// TwinCAT 3 PLC project PLC
// ProgramVersion: 3.1.4024.0
// libraries:
//   Tc2_Standard, * (Beckhoff Automation GmbH)
//   Tc2_System, * (Beckhoff Automation GmbH)
//   Tc2_Utilities, * (Beckhoff Automation GmbH)
//   Tc3_JsonXml, * (Beckhoff Automation GmbH)
//   Tc3_Module, * (Beckhoff Automation GmbH)
// project tree:
//   / FB_DynamicArrayBase64.TcPOU, FB_DynamicArrayBinary.TcPOU, FB_DynamicArrayOfLREAL.TcPOU, FB_DynamicArrayOfInt.TcPOU, MAIN.TcPOU, PlcTask.TcTTO
//   Test/ FB_Test.TcPOU, I_Test.TcIO
//   Utilities/ FB_TimeLimitedIterator.TcPOU
// real-time tasks:
//   TASK PlcTask: cycle T#10ms, priority 20, ADS port 350

CONFIGURATION PLC
    RESOURCE PLC ON TwinCAT3
        TASK PlcTask(INTERVAL := T#10ms, PRIORITY := 20);
        PROGRAM MAIN WITH PlcTask : MAIN;
    END_RESOURCE
END_CONFIGURATION

// ---- Test/I_Test.TcIO
INTERFACE I_Test

METHOD METH : BOOL
VAR_INPUT
END_VAR
END_METHOD

PROPERTY Name : String
GET
END_GET
END_PROPERTY

END_INTERFACE

// ---- MAIN.TcPOU
PROGRAM MAIN
VAR
	aArray : FB_DynamicArrayBase64;
	bRemoveLast: BOOL;
	bRemoveFirst : BOOL;
	bRemoveIndex : BOOL;
	
	bAddTest : BOOL;
	bAddTestLoop : BOOL;
	bClear : BOOL;
	
	bSetIndex : BOOL;
END_VAR
VAR
	//=============================
	// Remove Index Test
	RemoveIndex : UDINT;
	
	//=============================
	// Set Inex Test
	nSetIndex : UDINT;
	//=============================
	// Add Test
	WriteBool : BOOL;
	WriteReal : LREAL;
	WriteString : STRING;
	
	iTest : I_Test;
	fbTest : FB_Test;
	
	//=============================
	// Add Test Loop
	nAddTest : INT := 1000;
	i : INT;
	sTest : STRING(32766);
	
	ArrayElements : UDINT;
	
	
	//==================================================
	//Get
	ReadBOOL : BOOL;
	ReadReal : LREAL;
	ReadString : STRING;
	ReadInterface : I_Test;
	
	bReadBOOL : BOOL;
	bReadREAL : BOOL;
	bReadString : BOOL;
	bReadInterface : BOOL;
	ReadIndex : UDINT;
	//==================================================
	//Time
	fbTimeLimitedIterator : FB_TimeLimitedIterator := (TaskUsagePercent := 100);
	ReadTime : LTIME;
	
	aTime : ARRAY[0..100000] OF LINT;
	aLREAL : FB_DynamicArrayOfINT;
	nTestLoop : UDINT := 10000;
	f : UDINT;
	fReadWrite : LINT;
	
	tTimeWriteArray : LTIME;
	tTimeReadArray : LTIME;
	
	tTimeAddDynamicArray : LTIME;
	tTimeWriteDynamicArray : LTIME;
	tTimeReadDynamicArray : LTIME;
	
	WriteFaktor : LREAL;
	ReadFaktor : LREAL;
END_VAR

ArrayElements := aArray.Count;
iTest := fbTest;

//=============================
// Add Test
IF bAddTest THEN
	bAddTest := FALSE;	
	aArray.AddLast(WriteBool);
	aArray.AddLast(WriteReal);
	aArray.AddStringLast(WriteString);
	aArray.AddLast(iTest);
END_IF

//=============================
// Add Test
IF bSetIndex THEN
	bSetIndex := FALSE;	
	aArray.TrySetIndex(nSetIndex, WriteBool);

END_IF
//=============================
// Add Test Loop
	IF bAddTestLoop THEN
		bAddTestLoop := FALSE;
		IF nAddTest > 0 THEN
			FOR i := 0 TO nAddTest - 1 DO
				aArray.AddLast(WriteBool);
				aArray.AddLast(WriteReal);
				aArray.AddStringLast(WriteString);
				aArray.AddLast(iTest);
			END_FOR
		END_IF
	END_IF

//=============================
// Clear
	IF bClear THEN
		bClear := FALSE;
		aArray.Clear();
	END_IF

//=============================
// Remove
	IF bRemoveLast THEN
		bRemoveLast := FALSE;
		aArray.RemoveLast();
	END_IF
	IF bRemoveFirst THEN
		bRemoveFirst := FALSE;
		aArray.RemoveFirst();
	END_IF
	IF bRemoveIndex THEN
		bRemoveIndex := FALSE;
		aArray.TryDeleteIndex(RemoveIndex);
	END_IF
	
//==================================================
//Get

	fbTimeLimitedIterator.SetIterationStartTime();
	
	bReadBOOL := aArray.TryGetIndex(ReadIndex,ReadBool);
	bReadREAL := aArray.TryGetIndex(ReadIndex,ReadReal);
	bReadString := aArray.TryGetIndex(ReadIndex,ReadString);
	bReadInterface := aArray.TryGetIndex(ReadIndex, ReadInterface);
	
	ReadTime := fbTimeLimitedIterator.CurrentIterationTime();

//==========================================================
// Debug String
	aArray.CopyArrayString(pDoc:= sTest, nDoc := SIZEOF(sTest));
	
//==========================================================
// Timing Test
	nTestLoop := LIMIT(0,nTestLoop ,100000);
	
	fbTimeLimitedIterator.SetIterationStartTime();
		FOR f := 0 TO nTestLoop DO
			aTime[f] := fReadWrite;
		END_FOR
	tTimeWriteArray := fbTimeLimitedIterator.CurrentIterationTime();
	
	
	fbTimeLimitedIterator.SetIterationStartTime();
		FOR f := 0 TO nTestLoop DO
			fReadWrite := aTime[f];
		END_FOR
	tTimeReadArray := fbTimeLimitedIterator.CurrentIterationTime();
	

	
	aLREAL.Clear();
	
	fbTimeLimitedIterator.SetIterationStartTime();
		FOR f := 0 TO nTestLoop DO
			aLREAL.AddLast(fReadWrite);
		END_FOR
	tTimeAddDynamicArray := fbTimeLimitedIterator.CurrentIterationTime();
	
	fbTimeLimitedIterator.SetIterationStartTime();
		FOR f := 0 TO nTestLoop DO
			aLREAL.TrySetIndex(f,fReadWrite);
		END_FOR
	tTimeWriteDynamicArray := fbTimeLimitedIterator.CurrentIterationTime();
	
	fbTimeLimitedIterator.SetIterationStartTime();
		FOR f := 0 TO nTestLoop DO
			aLREAL.TryGetIndex(f,fReadWrite);
		END_FOR
	tTimeReadDynamicArray := fbTimeLimitedIterator.CurrentIterationTime();

	
	
	IF tTimeReadArray <> LTIME#0S THEN
		ReadFaktor := TO_LREAL(TO_LREAL(tTimeReadDynamicArray*10000)/TO_LREAL(tTimeReadArray*10000));
	END_IF
	IF tTimeWriteArray <> LTIME#0S THEN
		WriteFaktor := TO_LREAL(TO_LREAL(tTimeWriteDynamicArray*10000)/TO_LREAL( tTimeWriteArray*10000));
	END_IF

END_PROGRAM

// ---- FB_DynamicArrayBase64.TcPOU
{attribute 'no_explicit_call' := 'This FB is a CLASS and must be accessed using methods or properties'}
{attribute 'enable_dynamic_creation'}
{attribute 'hide_all_locals'}
FUNCTION_BLOCK FB_DynamicArrayBase64
VAR
	buffer : FB_JsonDynDomParser;
	root : sJsonValue;
END_VAR

PROPERTY PRIVATE _Array : sJsonValue
GET
IF root <> 0 THEN
	_Array := root;
ELSE
	root := buffer.NewDocument();
	_Array := buffer.SetArray(root,0);
END_IF
END_GET
END_PROPERTY

METHOD PUBLIC AddLast : BOOL
VAR_INPUT
	Value : ANY;
END_VAR
AddLast := buffer.PushbackBase64Value(v:= _Array, p := Value.pValue,n := Value.diSize) <> 0;
END_METHOD

METHOD PUBLIC AddStringLast : BOOL
VAR_INPUT
	Value : ANY_STRING;
END_VAR
AddStringLast := buffer.PushbackBase64Value(v:= _Array, p := Value.pValue,n := TO_DINT(LEN2(Value.pValue)+ 1)) <> 0;
END_METHOD

METHOD PUBLIC Clear : BOOL
VAR
	_arrayElement : SJsonAIterator;
END_VAR
_arrayElement := buffer.ArrayBegin(_array);
IF _arrayElement <> 0 THEN
	Clear := buffer.ClearArray(v := _array,i := _arrayElement);
END_IF
END_METHOD

METHOD PUBLIC CopyArrayString : BOOL
VAR_IN_OUT CONSTANT
  	pDoc : STRING; 
END_VAR
VAR_INPUT
	nDoc : UDINT;
END_VAR
CopyArrayString := buffer.copyjson(v:= _Array, pDoc:= pDoc,nDoc := nDoc) <> 0;
END_METHOD

PROPERTY PUBLIC Count : UDINT
GET
Count := buffer.GetArraySize(_array);
END_GET
END_PROPERTY

PROPERTY PUBLIC FirstIndex : UDINT
GET
FirstIndex := 0;
END_GET
END_PROPERTY

PROPERTY PUBLIC LastIndex : UDINT
GET
IF Count = 0 THEN
	LastIndex := 0;
ELSE 
	LastIndex := Count - 1;
END_IF
END_GET
END_PROPERTY

METHOD PUBLIC RemoveFirst : BOOL
VAR
	_arrayElement : SJsonAIterator;
END_VAR
RemoveFirst := TryDeleteIndex(0);
END_METHOD

METHOD PUBLIC RemoveLast: BOOL
VAR
	_arrayElement : SJsonAIterator;
END_VAR
RemoveLast := TryDeleteIndex(LastIndex);
END_METHOD

METHOD PUBLIC TryDeleteIndex : BOOL
VAR_INPUT
	Index : UDINT;
END_VAR
VAR
	_arrayElement : SJsonAIterator;
END_VAR
_arrayElement := buffer.GetArrayValueByIdx(_Array, Index);
IF _arrayElement <> 0 THEN
	TryDeleteIndex := buffer.RemoveArray(v := _array,i := _arrayElement);
END_IF
END_METHOD

METHOD PUBLIC TryGetIndex : BOOL;
VAR_INPUT
	Index : UDINT;
	Destination : ANY;
END_VAR
TryGetIndex := buffer.GetBase64(v:=  buffer.GetArrayValueByIdx(_Array, Index),p := Destination.pValue, n:= Destination.diSize) <> 0;
END_METHOD

METHOD PUBLIC TryGetIndexTo : BOOL;
VAR_INPUT
	Index : UDINT;
	Destination : PVOID;
	DestinationSize : UDINT;
END_VAR
VAR
	_arrayElement : SJsonAIterator;
END_VAR
_arrayElement := buffer.GetArrayValueByIdx(_Array, Index);
IF _arrayElement <> 0 THEN
	TryGetIndexTo := buffer.GetBase64(v:= _arrayElement,p := Destination, n:= TO_DINT(DestinationSize)) <> 0;
END_IF
END_METHOD

METHOD PUBLIC TrySetIndex : BOOL
VAR_INPUT
	Index : UDINT;
	Value : ANY;
END_VAR
TrySetIndex := buffer.SetBase64(v:= buffer.GetArrayValueByIdx(_Array, Index),p := Value.pValue, n:= Value.diSize) <> 0;
END_METHOD

METHOD PUBLIC TrySetIndexTo : BOOL
VAR_INPUT
	Index : UDINT;
	Value : PVOID;
	ValueSize : UDINT;
END_VAR
VAR
	_arrayElement : SJsonAIterator;
END_VAR
_arrayElement := buffer.GetArrayValueByIdx(_Array, Index);
IF _arrayElement <> 0 THEN
	TrySetIndexTo := buffer.SetBase64(v:= _arrayElement,p := Value, n:= TO_DINT(ValueSize)) <> 0;
END_IF
END_METHOD

END_FUNCTION_BLOCK

// ---- Test/FB_Test.TcPOU
FUNCTION_BLOCK FB_Test IMPLEMENTS I_Test
VAR_INPUT
END_VAR
VAR_OUTPUT
END_VAR
VAR
END_VAR

METHOD METH : BOOL
VAR_INPUT
END_VAR
END_METHOD

PROPERTY Name : STRING
GET
Name := 'Test';
END_GET
END_PROPERTY

END_FUNCTION_BLOCK

// ---- Utilities/FB_TimeLimitedIterator.TcPOU
FUNCTION_BLOCK FB_TimeLimitedIterator
VAR
    nLocalTaskUsagePercent : BYTE; 
    fbGetTickTime : GETCPUCOUNTER;
    TaskIndex : DINT;
    
    nInterruptThreshold : UDINT;
    nLocalCycleTime : UDINT;
    nIterationStartTime : ULINT;
    nIterationCurrentTime : ULINT;
    nIterationElapsedTime : UDINT;
END_VAR

METHOD PUBLIC CheckInterationTimeExceeded : BOOL
VAR_INPUT
END_VAR
fbGetTickTime();

nIterationCurrentTime := DWORD_TO_ULINT(fbGetTickTime.cpuCntLoDW) OR SHL(DWORD_TO_ULINT(fbGetTickTime.cpuCntHiDW), 32);
nIterationElapsedTime := ULINT_TO_UDINT (THIS^.nIterationCurrentTime - THIS^.nIterationStartTime);

CheckInterationTimeExceeded := nIterationElapsedTime >= nInterruptThreshold;
END_METHOD

METHOD CurrentIterationTime : LTIME
VAR
    CurrentTime : ULINT;
END_VAR
fbGetTickTime();

CurrentTime := DWORD_TO_ULINT(fbGetTickTime.cpuCntLoDW) OR SHL(DWORD_TO_ULINT(fbGetTickTime.cpuCntHiDW), 32);

CurrentIterationTime := ULINT_TO_LTIME (CurrentTime - THIS^.nIterationStartTime)*100;
END_METHOD

METHOD PUBLIC SetIterationStartTime : BOOL
VAR_INPUT
END_VAR
IF TaskIndex = 0 OR TaskIndex <> GETCURTASKINDEXEX() THEN
    TaskIndex := GETCURTASKINDEXEX();
    nLocalCycleTime := TwinCAT_SystemInfoVarList._TaskInfo[TaskIndex].CycleTime;
    nInterruptThreshold:= (nLocalCycleTime * LIMIT(1, TaskUsagePercent, 100)) / 100;
END_IF

fbGetTickTime();
nIterationStartTime := DWORD_TO_ULINT(fbGetTickTime.cpuCntLoDW) OR SHL(DWORD_TO_ULINT(fbGetTickTime.cpuCntHiDW), 32);
END_METHOD

PROPERTY PUBLIC TaskUsagePercent : BYTE
GET
TaskUsagePercent := nLocalTaskUsagePercent;
END_GET
SET
IF nLocalTaskUsagePercent <> TaskUsagePercent THEN
    nLocalTaskUsagePercent := TaskUsagePercent;
    
    TaskIndex := GETCURTASKINDEXEX();
	IF TaskIndex <> 0 THEN
		nLocalCycleTime := TwinCAT_SystemInfoVarList._TaskInfo[TaskIndex].CycleTime;
   	 	nInterruptThreshold:= (nLocalCycleTime * LIMIT(1, TaskUsagePercent, 100)) / 100;
	END_IF
END_IF
END_SET
END_PROPERTY

END_FUNCTION_BLOCK

// ---- FB_DynamicArrayOfInt.TcPOU
{attribute 'no_explicit_call' := 'This FB is a CLASS and must be accessed using methods or properties'}
{attribute 'enable_dynamic_creation'}
//{attribute 'hide_all_locals'}
FUNCTION_BLOCK FB_DynamicArrayOfInt
VAR
	buffer : FB_JsonDomParser;
	root : sJsonValue;
END_VAR

PROPERTY PRIVATE _Array : sJsonValue
GET
IF root <> 0 THEN
	_Array := root;
ELSE
	root := buffer.NewDocument();
	_Array := buffer.SetArray(root,0);
END_IF
END_GET
END_PROPERTY

METHOD PUBLIC AddLast : BOOL
VAR_IN_OUT
	Value : LINT;
END_VAR
AddLast := buffer.PushbackInt64Value(v:= _Array, Value) <> 0;
END_METHOD

METHOD PUBLIC Clear : BOOL
VAR
	_arrayElement : SJsonAIterator;
END_VAR
_arrayElement := buffer.ArrayBegin(_array);
IF _arrayElement <> 0 THEN
	Clear := buffer.ClearArray(v := _array,i := _arrayElement);
END_IF
END_METHOD

METHOD PUBLIC CopyArrayString : BOOL
VAR_IN_OUT CONSTANT
  	pDoc : STRING; 
END_VAR
VAR_INPUT
	nDoc : UDINT;
END_VAR
CopyArrayString := buffer.copyjson(v:= _Array, pDoc:= pDoc,nDoc := nDoc) <> 0;
END_METHOD

PROPERTY PUBLIC Count : UDINT
GET
Count := buffer.GetArraySize(_array);
END_GET
END_PROPERTY

PROPERTY PUBLIC FirstIndex : UDINT
GET
FirstIndex := 0;
END_GET
END_PROPERTY

PROPERTY PUBLIC LastIndex : UDINT
GET
IF Count = 0 THEN
	LastIndex := 0;
ELSE 
	LastIndex := Count - 1;
END_IF
END_GET
END_PROPERTY

METHOD PUBLIC RemoveFirst : BOOL
VAR
	_arrayElement : SJsonAIterator;
END_VAR
RemoveFirst := TryDeleteIndex(0);
END_METHOD

METHOD PUBLIC RemoveLast: BOOL
VAR
	_arrayElement : SJsonAIterator;
END_VAR
RemoveLast := TryDeleteIndex(LastIndex);
END_METHOD

METHOD PUBLIC TryDeleteIndex : BOOL
VAR_INPUT
	Index : UDINT;
END_VAR
VAR
	_arrayElement : SJsonAIterator;
END_VAR
_arrayElement := buffer.GetArrayValueByIdx(_Array, Index);
IF _arrayElement <> 0 THEN
	TryDeleteIndex := buffer.RemoveArray(v := _array,i := _arrayElement);
END_IF
END_METHOD

METHOD PUBLIC TryGetIndex : BOOL;
VAR_INPUT
	Index : UDINT;	
END_VAR
VAR_IN_OUT
	Destination : LINT;
END_VAR
Destination := buffer.GetInt64(v:= buffer.GetArrayValueByIdx(_Array, Index));
END_METHOD

METHOD PUBLIC TrySetIndex : BOOL
VAR_INPUT
	Index : UDINT;
END_VAR
VAR_IN_OUT
	Value : LINT;
END_VAR
TrySetIndex := buffer.SetInt64(v:= buffer.GetArrayValueByIdx(_Array, Index),Value) <> 0;
END_METHOD

END_FUNCTION_BLOCK

// ---- FB_DynamicArrayBinary.TcPOU
{attribute 'no_explicit_call' := 'This FB is a CLASS and must be accessed using methods or properties'}
{attribute 'enable_dynamic_creation'}
{attribute 'hide_all_locals'}
FUNCTION_BLOCK FB_DynamicArrayBinary
VAR
	buffer : FB_JsonDynDomParser;
	root : sJsonValue;
END_VAR

PROPERTY PRIVATE _Array : sJsonValue
GET
IF root <> 0 THEN
	_Array := root;
ELSE
	root := buffer.NewDocument();
	_Array := buffer.SetArray(root,0);
END_IF
END_GET
END_PROPERTY

METHOD PUBLIC AddLast : BOOL
VAR_INPUT
	Value : ANY;
END_VAR
AddLast := buffer.PushbackHexBinaryValue(v:= _Array, p := Value.pValue,n := Value.diSize) <> 0;
END_METHOD

METHOD PUBLIC AddStringLast : BOOL
VAR_INPUT
	Value : ANY_STRING;
END_VAR
AddStringLast := buffer.PushbackHexBinaryValue(v:= _Array, p := Value.pValue,n := TO_DINT(LEN2(Value.pValue)+ 1)) <> 0;
END_METHOD

METHOD PUBLIC Clear : BOOL
VAR
	_arrayElement : SJsonAIterator;
END_VAR
_arrayElement := buffer.ArrayBegin(_array);
IF _arrayElement <> 0 THEN
	Clear := buffer.ClearArray(v := _array,i := _arrayElement);
END_IF
END_METHOD

METHOD PUBLIC CopyArrayString : BOOL
VAR_IN_OUT CONSTANT
  	pDoc : STRING; 
END_VAR
VAR_INPUT
	nDoc : UDINT;
END_VAR
CopyArrayString := buffer.copyjson(v:= _Array, pDoc:= pDoc,nDoc := nDoc) <> 0;
END_METHOD

PROPERTY PUBLIC Count : UDINT
GET
Count := buffer.GetArraySize(_array);
END_GET
END_PROPERTY

PROPERTY PUBLIC FirstIndex : UDINT
GET
FirstIndex := 0;
END_GET
END_PROPERTY

PROPERTY PUBLIC LastIndex : UDINT
GET
IF Count = 0 THEN
	LastIndex := 0;
ELSE 
	LastIndex := Count - 1;
END_IF
END_GET
END_PROPERTY

METHOD PUBLIC RemoveFirst : BOOL
VAR
	_arrayElement : SJsonAIterator;
END_VAR
RemoveFirst := TryDeleteIndex(0);
END_METHOD

METHOD PUBLIC RemoveLast: BOOL
VAR
	_arrayElement : SJsonAIterator;
END_VAR
RemoveLast := TryDeleteIndex(LastIndex);
END_METHOD

METHOD PUBLIC TryDeleteIndex : BOOL
VAR_INPUT
	Index : UDINT;
END_VAR
VAR
	_arrayElement : SJsonAIterator;
END_VAR
_arrayElement := buffer.GetArrayValueByIdx(_Array, Index);
IF _arrayElement <> 0 THEN
	TryDeleteIndex := buffer.RemoveArray(v := _array,i := _arrayElement);
END_IF
END_METHOD

METHOD PUBLIC TryGetIndex : BOOL;
VAR_INPUT
	Index : UDINT;
	Destination : ANY;
END_VAR
	TryGetIndex := buffer.GetHexBinary(v:=  buffer.GetArrayValueByIdx(_Array, Index),p := Destination.pValue, n:= Destination.diSize) <> 0;
END_METHOD

METHOD PUBLIC TryGetIndexTo : BOOL;
VAR_INPUT
	Index : UDINT;
	Destination : PVOID;
	DestinationSize : UDINT;
END_VAR
VAR
	_arrayElement : SJsonAIterator;
END_VAR
_arrayElement := buffer.GetArrayValueByIdx(_Array, Index);
IF _arrayElement <> 0 THEN
	TryGetIndexTo := buffer.GetHexBinary(v:= _arrayElement,p := Destination, n:= TO_DINT(DestinationSize)) <> 0;
END_IF
END_METHOD

METHOD PUBLIC TrySetIndex : BOOL
VAR_INPUT
	Index : UDINT;
	Value : ANY;
END_VAR
TrySetIndex := buffer.SetHexBinary(v:= buffer.GetArrayValueByIdx(_Array, Index),p := Value.pValue, n:= Value.diSize) <> 0;
END_METHOD

METHOD PUBLIC TrySetIndexTo : BOOL
VAR_INPUT
	Index : UDINT;
	Value : PVOID;
	ValueSize : UDINT;
END_VAR
VAR
	_arrayElement : SJsonAIterator;
END_VAR
_arrayElement := buffer.GetArrayValueByIdx(_Array, Index);
IF _arrayElement <> 0 THEN
	TrySetIndexTo := buffer.SetHexBinary(v:= _arrayElement,p := Value, n:= TO_DINT(ValueSize)) <> 0;
END_IF
END_METHOD

END_FUNCTION_BLOCK

// ---- FB_DynamicArrayOfLREAL.TcPOU
{attribute 'no_explicit_call' := 'This FB is a CLASS and must be accessed using methods or properties'}
{attribute 'enable_dynamic_creation'}
//{attribute 'hide_all_locals'}
FUNCTION_BLOCK FB_DynamicArrayOfLREAL
VAR
	buffer : FB_JsonDomParser;
	root : sJsonValue;
END_VAR

PROPERTY PRIVATE _Array : sJsonValue
GET
IF root <> 0 THEN
	_Array := root;
ELSE
	root := buffer.NewDocument();
	_Array := buffer.SetArray(root,0);
END_IF
END_GET
END_PROPERTY

METHOD PUBLIC AddLast : BOOL
VAR_IN_OUT
	Value : LREAL;
END_VAR
AddLast := buffer.PushbackDoubleValue(v:= _Array, Value) <> 0;
END_METHOD

METHOD PUBLIC Clear : BOOL
VAR
	_arrayElement : SJsonAIterator;
END_VAR
_arrayElement := buffer.ArrayBegin(_array);
IF _arrayElement <> 0 THEN
	Clear := buffer.ClearArray(v := _array,i := _arrayElement);
END_IF
END_METHOD

METHOD PUBLIC CopyArrayString : BOOL
VAR_IN_OUT CONSTANT
  	pDoc : STRING; 
END_VAR
VAR_INPUT
	nDoc : UDINT;
END_VAR
CopyArrayString := buffer.copyjson(v:= _Array, pDoc:= pDoc,nDoc := nDoc) <> 0;
END_METHOD

PROPERTY PUBLIC Count : UDINT
GET
Count := buffer.GetArraySize(_array);
END_GET
END_PROPERTY

PROPERTY PUBLIC FirstIndex : UDINT
GET
FirstIndex := 0;
END_GET
END_PROPERTY

PROPERTY PUBLIC LastIndex : UDINT
GET
IF Count = 0 THEN
	LastIndex := 0;
ELSE 
	LastIndex := Count - 1;
END_IF
END_GET
END_PROPERTY

METHOD PUBLIC RemoveFirst : BOOL
VAR
	_arrayElement : SJsonAIterator;
END_VAR
RemoveFirst := TryDeleteIndex(0);
END_METHOD

METHOD PUBLIC RemoveLast: BOOL
VAR
	_arrayElement : SJsonAIterator;
END_VAR
RemoveLast := TryDeleteIndex(LastIndex);
END_METHOD

METHOD PUBLIC TryDeleteIndex : BOOL
VAR_INPUT
	Index : UDINT;
END_VAR
VAR
	_arrayElement : SJsonAIterator;
END_VAR
_arrayElement := buffer.GetArrayValueByIdx(_Array, Index);
IF _arrayElement <> 0 THEN
	TryDeleteIndex := buffer.RemoveArray(v := _array,i := _arrayElement);
END_IF
END_METHOD

METHOD PUBLIC TryGetIndex : BOOL;
VAR_INPUT
	Index : UDINT;	
END_VAR
VAR_IN_OUT
	Destination : LREAL;
END_VAR
Destination := buffer.GetDouble(v:= buffer.GetArrayValueByIdx(_Array, Index));
END_METHOD

METHOD PUBLIC TrySetIndex : BOOL
VAR_INPUT
	Index : UDINT;
END_VAR
VAR_IN_OUT
	Value : LREAL;
END_VAR
TrySetIndex := buffer.SetDouble(v:= buffer.GetArrayValueByIdx(_Array, Index),Value) <> 0;
END_METHOD

END_FUNCTION_BLOCK
